{attribute 'GeneratedUsingTerminal: CU1128--0000'}
{attribute addProperty BoxType "CU1128--0000"}
{attribute addProperty Id "A_0005_CU1128_0000_0001A_0005_CU1128_0000_0001_8DEFD527120A_0004_CU1128_0000_0000_2_CU1128_BCU1128_1FC0878B2A_0004_CU1128_0000_0000_3_CU1128_CCU1128_1FC0878B2"}
{attribute addProperty CRC "794876575"}
{attribute addProperty Size "124"}
TYPE A_0004_CU1128_0000_0000_2F60DA9F EXTENDS CU1128_1FC0878B :
STRUCT
	{attribute addProperty Name "A_0005_CU1128_0000_0001"}
	{attribute addProperty PreviousPort "A_0004(CU1128-0000-0000) : D"}
	A_0005_CU1128_0000_0001 : A_0005_CU1128_0000_0001_8DEFD527;
	{attribute addProperty Name "A_0004_CU1128_0000_0000_2_CU1128_B"}
	{attribute addProperty PreviousPort "A_0004(CU1128-0000-0000) : C"}
	A_0004_CU1128_0000_0000_2_CU1128_B : CU1128_1FC0878B;
	{attribute addProperty Name "A_0004_CU1128_0000_0000_3_CU1128_C"}
	{attribute addProperty PreviousPort "A_0004(CU1128-0000-0000)_2 (CU1128-B) : C"}
	A_0004_CU1128_0000_0000_3_CU1128_C : CU1128_1FC0878B;
END_STRUCT
END_TYPE

(* stored: Version 1.2.0.0, ProductVersion 3.1.4024.9
   DUT A_0004_CU1128_0000_0000_2F60DA9F: Id {d52ab9cf-d0ce-4f7f-af01-b90c2b2fbaac} *)
